(* PLC project Safety, BrAutomation SafeDESIGNER  5.23.0.0 *)
(* stored: companyURL http://www.br-automation.com, creationDateTime Mon Aug 21 13:44:54 2023 *)

PROGRAM Main

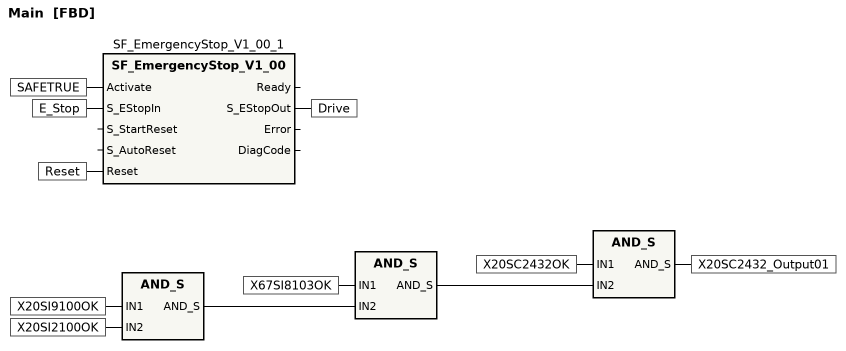
(* FBD diagram, written out as Structured Text *)
SF_EmergencyStop_V1_00_1(Activate := SAFETRUE, S_EStopIn := E_Stop, Reset := Reset);
Drive := SF_EmergencyStop_V1_00_1.S_EStopOut;
X20SC2432_Output01 := AND_S(X20SC2432OK, AND_S(X67SI8103OK, AND_S(X20SI9100OK, X20SI2100OK)));
END_PROGRAM
